TYPE IOExpantionMessageErrorEx_t :
STRUCT
	isErrorActive : BOOL := FALSE; // a variable to attach to primitiveWatchdogHandler
	errorMessageCallback : BOOL := FALSE; // callback for IOExpantionHandler_t
	clearMessageCallback : BOOL := FALSE; // callback for IOExpantionHandler_t
END_STRUCT
END_TYPE

(* stored: Version 1.1.0.1
   DUT IOExpantionMessageErrorEx_t: Id {4521a644-3825-48a5-b917-97d2d4d81dc4} *)
